FUNCTION_BLOCK Kims_UpdateLights
VAR_INPUT
	Intersect:POINTER TO Intersection;
	NightMode:BOOL;
END_VAR
VAR_OUTPUT
END_VAR
VAR
	LightState: (NS_Flow, EW_Flow, NorthOnly, SouthOnly, EastOnly, WestOnly, NS_Night, EW_Night);
	Transition:(NewLightState,To_Yellow,To_Red,To_Green, Stay_Green);
	TransitionTimer, FlowTimer,Blinktimer,PedWarning:TON;
	StayGreenTime:TIME:= T#40S;
END_VAR
VAR CONSTANT
	RED:INT:=0;
	AMBER:INT:=1;
	GREEN:INT:=2;
END_VAR

BlinkTimer(In:= NOT BlinkTimer.Q, PT:=(T#1S));
PedWarning(In:= NOT PedWarning.Q, PT:=(T#1S));

IF NightMode AND Intersect^.EW_Road >= Intersect^.NS_Road THEN
	LightState:= EW_Night;
ELSIF NightMode AND Intersect^.EW_Road < Intersect^.NS_Road THEN
	LightState:= NS_Night;
ELSIF LightState = NS_Flow AND Transition = NewLightState THEN
	LightState:= EW_Flow;
	Transition:=To_Yellow;
ELSIF LightState = EW_Flow AND Transition = NewLightState THEN
	LightState:= NS_Flow;
	Transition:=To_Yellow;
END_IF


CASE LightState OF
	NS_Flow:
		IF Intersect^.N_Ped OR Intersect^.S_Ped THEN
			Intersect^.N_Cross:=Intersect^.N_Ped;
			Intersect^.S_Cross:= Intersect^.S_Ped;
			StayGreenTime:= MAX(FlowTimer.ET+T#2S,T#10S) ;
		END_IF
		CASE Transition OF
			To_Yellow:
				Intersect^.E_Light.Amber:=TRUE;
				Intersect^.E_Light.Red := Intersect^.E_Light.Green:= FALSE;
				Intersect^.W_Light.Amber:=TRUE;
				Intersect^.W_Light.Red := Intersect^.W_Light.Green:= FALSE;
				TransitionTimer(IN:=NOT TransitionTimer.Q,PT:=(T#20S / Intersect^.EW_Road));
				IF TransitionTimer.Q THEN
				Transition:= To_Red;
				END_IF;	
			To_Red:
				Intersect^.E_Light.Red:=TRUE;
				Intersect^.E_Light.Amber := Intersect^.E_Light.Green:= FALSE;
				Intersect^.W_Light.Red:=TRUE;
				Intersect^.W_Light.Amber := Intersect^.W_Light.Green:= FALSE;
				TransitionTimer(IN:=NOT TransitionTimer.Q,PT:=(T#5S / Intersect^.EW_Road));
				IF TransitionTimer.Q THEN
				Transition:= To_Green;
				END_IF;
			To_Green:
				Intersect^.N_Light.Green:=TRUE;
				Intersect^.N_Light.Red := Intersect^.N_Light.Amber:= FALSE;
				Intersect^.S_Light.Green:=TRUE;
				Intersect^.S_Light.Red := Intersect^.S_Light.Amber:= FALSE;
				TransitionTimer(IN:=NOT TransitionTimer.Q,PT:=(T#2S));
				IF TransitionTimer.Q THEN
				Transition:= Stay_Green;
				END_IF;	
			Stay_Green:
				FlowTimer(In:= NOT FlowTimer.Q, PT:=(StayGreenTime / Intersect^.EW_Road));
				IF(FlowTimer.PT - FlowTimer.ET < T#5S) THEN
					IF PedWarning.Q THEN
						Intersect^.E_Cross:=Intersect^.W_Cross:= NOT Intersect^.E_Cross;
					END_IF
				ELSE
					Intersect^.E_Cross:=Intersect^.W_Cross:= TRUE;
				END_IF
				IF FlowTimer.Q THEN
				Transition:= NewLightState;
				END_IF;	
		END_CASE
	EW_Flow:
		IF Intersect^.E_Ped OR Intersect^.W_Ped THEN
			Intersect^.E_Cross:=Intersect^.E_Ped;
			Intersect^.W_Cross:= Intersect^.W_Ped;
			StayGreenTime:= MAX(FlowTimer.ET+T#2S,T#10S) ;
		END_IF
		CASE Transition OF
			To_Yellow:
				Intersect^.N_Light.Amber:=TRUE;
				Intersect^.N_Light.Red := Intersect^.N_Light.Green:= FALSE;
				Intersect^.S_Light.Amber:=TRUE;
				Intersect^.S_Light.Red := Intersect^.S_Light.Green:= FALSE;
				TransitionTimer(IN:=NOT TransitionTimer.Q,PT:=(T#20S / Intersect^.NS_Road));
				IF TransitionTimer.Q THEN
				Transition:= To_Red;
				END_IF;	
			To_Red:
				Intersect^.N_Light.Red:=TRUE;
				Intersect^.N_Light.Amber := Intersect^.N_Light.Green:= FALSE;
				Intersect^.S_Light.Red:=TRUE;
				Intersect^.S_Light.Amber:= Intersect^.S_Light.Green:= FALSE;
				TransitionTimer(IN:=NOT TransitionTimer.Q,PT:=(T#5S / Intersect^.NS_Road));
				IF TransitionTimer.Q THEN
				Transition:= To_Green;
				END_IF;
			To_Green:
				Intersect^.E_Light.Green:=TRUE;
				Intersect^.E_Light.Red := Intersect^.E_Light.Amber:= FALSE;
				Intersect^.W_Light.Green:=TRUE;
				Intersect^.W_Light.Red := Intersect^.W_Light.Amber:= FALSE;
				TransitionTimer(IN:=NOT TransitionTimer.Q,PT:=(T#2S));
				IF TransitionTimer.Q THEN
				Transition:= Stay_Green;
				END_IF;				

Transition:= Stay_Green;
			Stay_Green:
				FlowTimer(In:= NOT FlowTimer.Q, PT:=(StayGreenTime / Intersect^.EW_Road));
				IF(FlowTimer.PT - FlowTimer.ET < T#5S) THEN
					IF PedWarning.Q THEN
						Intersect^.N_Cross:=Intersect^.S_Cross:= NOT Intersect^.N_Cross;
					END_IF
				ELSE
					Intersect^.N_Cross:=Intersect^.S_Cross:= TRUE;
				END_IF
				IF FlowTimer.Q THEN
				Transition:= NewLightState;
				END_IF;	
		END_CASE
	NorthOnly:
	
	SouthOnly:
	
	EastOnly:
	
	WestOnly:
	
	NS_Night:		
			;
			IF BlinkTimer.Q THEN
			Intersect^.N_Light.Amber:=Intersect^.S_Light.Amber:= NOT Intersect^.N_Light.Amber;
			Intersect^.E_Light.Red:=Intersect^.W_Light.Red:= NOT Intersect^.E_Light.Red;
			END_IF;
			Transition:= NewLightState;
	EW_Night:
			
			IF BlinkTimer.Q THEN
			Intersect^.E_Light.Amber:=Intersect^.W_Light.Amber:= NOT Intersect^.E_Light.Amber;
			Intersect^.N_Light.Red:=Intersect^.S_Light.Red:= NOT Intersect^.N_Light.Red;
			END_IF;
			Transition:= NewLightState;
END_CASE

METHOD SetLight : BOOL
VAR_INPUT
	Light: POINTER TO TrafficLight;
	Setting: INT;
END_VAR
CASE Setting OF
	RED:
	Light^.Red:=TRUE;
	Light^.Amber := Light^.Green:= FALSE;
	AMBER:
	Light^.Amber:=TRUE;
	Light^.Red := Light^.Green:= FALSE;
	GREEN:
	Light^.Green:=TRUE;
	Light^.Amber := Light^.Red:= FALSE;
END_CASE
END_METHOD

END_FUNCTION_BLOCK

(* stored: Version 1.1.0.1, ProductVersion 3.1.4024.11
   POU Kims_UpdateLights: Id {17a4a239-a718-4f43-ac46-8ffcc4f9c047}, SpecialFunc None
   Method SetLight: Id {f45c2384-f701-47b6-aeee-55db2e125d4c} *)
